FUNCTION_BLOCK ObservePAC EXTENDS HardwareObservationBase
VAR_INPUT
END_VAR
VAR_OUTPUT
END_VAR
VAR
	m_ptrPAC: POINTER TO PicAlphaConveyor;
	m_ptrPACWP1: POINTER TO xPPUProduct;
	m_ptrPACWP2: POINTER TO xPPUProduct;
	m_ptrPACWP3: POINTER TO xPPUProduct;
END_VAR

METHOD FB_init : BOOL
VAR_INPUT
	bInitRetains : BOOL; // if TRUE, the retain variables are initialized (warm start / cold start)
	bInCopyCode : BOOL;  // if TRUE, the instance afterwards gets moved into the copy code (online change)
	
	i_ptrPAC: POINTER TO PicAlphaConveyor;
	i_ptrWP1: POINTER TO xPPUProduct;
	i_ptrWP2: POINTER TO xPPUProduct;
	i_ptrWP3: POINTER TO xPPUProduct;

	
END_VAR
m_ptrPAC := i_ptrPAC;
m_ptrPACWP1 := i_ptrWP1;
m_ptrPACWP2 := i_ptrWP2;
m_ptrPACWP3 := i_ptrWP3;
END_METHOD

METHOD  ResetDefinition : BOOL
VAR_INPUT
END_VAR
;
END_METHOD

(* Update an instance of ProcessState with the part of the process that can be observed by this Hardware Interface. *)
METHOD UpdateProcessObservation : BOOL
VAR_IN_OUT
	io_processState: ProcessState;
END_VAR
io_processState.UpdateState_Binary(EProcessVariables.PAC_WPAtStart, m_ptrPAC^.WPAtStart, TRUE);
io_processState.UpdateState_Binary(EProcessVariables.PAC_WPAtEnd, m_ptrPAC^.WPAtEnd, TRUE);
io_processState.UpdateState_Binary(EProcessVariables.PAC_SwitchExtended, m_ptrPAC^.m_Switch.Extended, TRUE);
io_processState.UpdateState_Binary(EProcessVariables.PAC_SwitchRetracted, m_ptrPAC^.m_Switch.Retracted, TRUE);
io_processState.UpdateState_Numeric(EProcessVariables.PAC_WPNumber, INT_TO_LREAL(m_ptrPAC^.m_WPNumberAtPAC), TRUE);

io_processState.UpdateState_Defined(EProcessVariables.PAC_WPAtStart, TRUE);
io_processState.UpdateState_Defined(EProcessVariables.PAC_WPAtEnd, TRUE);
io_processState.UpdateState_Defined(EProcessVariables.PAC_SwitchExtended, TRUE);
io_processState.UpdateState_Defined(EProcessVariables.PAC_SwitchRetracted, TRUE);
io_processState.UpdateState_Defined(EProcessVariables.PAC_WPNumber, TRUE);
END_METHOD

END_FUNCTION_BLOCK

(* stored: Version 1.1.0.1
   POU ObservePAC: Id {f655d9cb-93c8-4fa4-b968-cd86aa308a91}, SpecialFunc None
   Method FB_init: Id {585d10f7-907a-460f-bb8b-74fb5484cb9b}
   Method ResetDefinition: Id {040df874-5fd1-4e6f-9865-9806b259212e}
   Method UpdateProcessObservation: Id {55b685a7-d601-4f6d-81ea-0d036a54c12c} *)
